VAR_GLOBAL
	// INPUT FISICI
Start        : BOOL;
Stop         : BOOL;
PieceSensor  : BOOL;
EStop        : BOOL;
InterlockOK  : BOOL;
Reset        : BOOL;

// OUTPUT FISICI
MotorOut      : BOOL;
ValveOpenOut  : BOOL;
ValveCloseOut : BOOL;

SimOpenFB  : BOOL;
SimCloseFB : BOOL;
SimMotorFB : BOOL;
END_VAR

(* stored: Version 1.1.0.1, ProductVersion 3.1.4024.16
   GVL GVL: Id {41ae355d-2b94-45c0-8937-6823f4319711} *)
